// TIA Portal V20 export
DATA_BLOCK "HMI_Central_Shifter"   // DB32
{ S7_Optimized_Access := 'TRUE' }
// stored: MemoryReserve 100
   VAR
      CS_PP_Reset : Bool;
      CS_PL_Reset : Bool;
      CS_TP_Reset : Bool;
      CS_TL_Reset : Bool;
      CS_Virtual_Reset : Bool;
      CS_Reset : Bool;
      CS_Homing : Bool;
      CS_PP_Power : Bool;
      CS_PL_Power : Bool;
      CS_TP_Power : Bool;
      CS_TL_Power : Bool;
      CS_Virtual_Power : Bool;
      CS_Power : Bool;
      CS_Gear_In : Bool;
      CS_Destination_Pos : Int := 7;
      CS_Drive_To_Des : Bool;
      CS_RL_Hydraulic_Up : Bool;
      CS_RL_Hydraulic_Down : Bool;
      CS_RP_Hydraulic_Up : Bool;
      CS_RP_Hydraulic_Down : Bool;
      CS_RL_Go_Forward : Bool;
      CS_RP_Go_Forward : Bool;
      CS_RP_Go_Backward : Bool;
      CS_RL_Go_Backward : Bool;
      CS_RL_RP_Reset : Bool;
      CS_Sides_Go_Up : Bool;
      CS_Sides_Go_Down : Bool;
      CS_Sides_Go_Mid : Bool;
      CS_Auto : Bool;
      CS_Side_Pos_Up : DInt;
      CS_Side_Pos_Mid : DInt;
      CS_Side_Pos_Down : DInt;
      CS_Pallet_Left_Move : Bool;
      CS_Pallet_Right_Move : Bool;
      CS_Pallet_Centering : Bool;
      CS_Go_Left : Bool;
      CS_Go_Right : Bool;
      CS_Auto_Hyd_Up : Bool;
      CS_Auto_Hyd_Down : Bool;
      CS_Reset_Hydro : Bool;
      CS_Auto_Pos_Start : Int;
      CS_Auto_Pos_End : Int;
      CS_Permission_Auto : Bool;
      CS_Status_Auto_Go_to_Des : SInt;
      Alarms : Word;   // PP/PL/TP/TL Power, GearIN, MoveVirtual
   END_VAR
BEGIN
END_DATA_BLOCK
